// TIA Portal V17 export
// export: Created 2023-12-22T15:08:06.1192638Z, ExportSetting WithDefaults, DisplayName Totally Integrated Automation Portal, DisplayVersion V17, DisplayName TIA Portal Openness, DisplayVersion V17, DisplayName TIA Portal Version Control Interface, DisplayVersion V17, DisplayName STEP 7 Professional, DisplayVersion V17, DisplayName STEP 7 Safety, DisplayVersion V17, DisplayName WinCC Advanced, DisplayVersion V17
DATA_BLOCK "PID_V_1_DB"   // DB903
VERSION : 0.1
// stored: AutoNumber false, DBAccessibleFromOPCUA true, DBAccessibleFromWebserver true, InstanceOfName PID_ex, InstanceOfType FB
"PID_ex"
   // VAR_INPUT
   //    Start : Bool;
   //    SP_A : Real;
   //    Value : Real;
   // END_VAR
   // VAR_OUTPUT
   //    PWM : Bool;
   //    Result : Real;
   // END_VAR
   // VAR_IN_OUT
   //    PID : PID_Compact;
   // END_VAR
   // VAR RETAIN
   //    CMD : "CMD";
   //    SP_M : Real;
   //    SP : Real;
   //    x { S7_SetPoint := 'True'} : Real := 1.0;
   //    SP_x : Real;
   //    Value_x : Real;
   //    Buffer : Real;
   //    PID_Output : Real;
   //    PID_Hand : Real;
   //    Sys : Struct
   //       Err_Ack : Bool;
   //       Alm_SP_H : Bool;
   //       Alm_SP_L : Bool;
   //       Alm_In_H : Bool;
   //       Alm_In_L : Bool;
   //       Activate : Bool;
   //       First_Run { S7_SetPoint := 'True'} : Bool := TRUE;
   //       Error_code : DWord;
   //       Warning_code : DWord;
   //       "Type" : Int;
   //       State : Int;
   //       Mode : Int;
   //    END_STRUCT;
   //    Settings : Struct
   //       SP_P { S7_SetPoint := 'True'} : Real := -1.5;
   //       SP_Ti { S7_SetPoint := 'True'} : Real := 150.0;
   //       SP_Td { S7_SetPoint := 'True'} : Real := 0.0;
   //       SP_Cycle { S7_SetPoint := 'True'} : Real := 0.2;
   //       Max_SP { S7_SetPoint := 'True'} : Real := 500.0;
   //       Min_SP { S7_SetPoint := 'True'} : Real := -500.0;
   //       Max_in { S7_SetPoint := 'True'} : Real := 500.0;
   //       Min_in { S7_SetPoint := 'True'} : Real := -500.0;
   //       Max_out { S7_SetPoint := 'True'} : Real := 100.0;
   //       Min_out { S7_SetPoint := 'True'} : Real := 0.0;
   //       DeadBand { S7_SetPoint := 'True'} : Real := 1.0;
   //       Max : Real;
   //       Min : Real;
   //    END_STRUCT;
   //    Converter : "Converter_LAD";
   //    Conveter_Back : "Converter_LAD";
   //    pos { S7_SetPoint := 'True'} : Array[0..15] of Bool;
   // END_VAR
BEGIN
   pos[0..15] := FALSE;
END_DATA_BLOCK
